// TIA Portal V20 export
TYPE "typeEmMotorStarterInterface"
// stored: Access Published
   STRUCT
      EMmotorstarter : Array[0.."NO_OF_EM"] of "typeMotorStarterInterface";
   END_STRUCT;
END_TYPE
